// TIA Portal project "Encoder _3" (V16)

(* hardware
DEVICE "S7-1200 station_1"  S7-1200 Station
   slot 0: "Rack_0"  S7-1200 Rack  Rack  V1.0
   slot 1: "PLC_1"  CPU 1212C DC/DC/DC  6ES7 212-1AE40-0XB0  V4.1
*)

// ===== PLC "PLC_1"  CPU 1212C DC/DC/DC =====

VAR_GLOBAL   // PLC tag table "Default tag table"
   "System_Byte" AT %MD2 : DInt;
   "FirstScan" AT %M1.0 : Bool;
   "DiagStatusUpdate" AT %M1.1 : Bool;
   "AlwaysTRUE" AT %M1.2 : Bool;
   "AlwaysFALSE" AT %M1.3 : Bool;
   "Clock_Byte" AT %MB0 : Byte;
   "Clock_10Hz" AT %M0.0 : Bool;
   "Clock_5Hz" AT %M0.1 : Bool;
   "Clock_2.5Hz" AT %M0.2 : Bool;
   "Clock_2Hz" AT %M0.3 : Bool;
   "Clock_1.25Hz" AT %M0.4 : Bool;
   "Clock_1Hz" AT %M0.5 : Bool;
   "Clock_0.625Hz" AT %M0.6 : Bool;
   "Clock_0.5Hz" AT %M0.7 : Bool;
   "encoder" AT %ID1000 : DInt;
   "Tag_2" AT %Q0.0 : Bool;
   "al_limite_atg" AT %Q0.1 : Bool;
   "Tag_4" AT %Q0.3 : Bool;
   "Tag_5" AT %I0.0 : Bool;
   "Tag_6" AT %I0.1 : Bool;
   "Tag_7" AT %I0.2 : Bool;
   "clock" AT %M255.5 : Bool;
   "time_et" AT %MD256 : Time;
   "numero_rotacao" AT %MW300 : Word;
   "time_pt" AT %MD200 : Time;
   "Tag_1" AT %ID100 : DWord;
END_VAR

VAR_GLOBAL   // PLC tag table "Tag table_1"
   "SLI_DETACH_event" AT %I0.3 : Bool;
END_VAR

TYPE "User_data_type_1"
   STRUCT
      Element_1 : Bool;
   END_STRUCT;
END_TYPE

DATA_BLOCK "Data_block_1"   // DB1
{ S7_Optimized_Access := 'TRUE' }
VERSION : 0.1
   VAR RETAIN
      valor_contagem : DInt;
   END_VAR
   VAR
      valor_referencia : DInt := 400;
      novo_valor : DInt;
   END_VAR
BEGIN
END_DATA_BLOCK

ORGANIZATION_BLOCK "Main"   // OB1, LAD, ProgramCycle
TITLE = "Main Program Sweep (Cycle)"
{ S7_Optimized_Access := 'TRUE' }
VERSION : 0.1
   VAR_INPUT
      Initial_Call : Bool;   // Initial call of this OB
      Remanence : Bool;   // =True, if remanent data are available
   END_VAR
   VAR_TEMP
      Temp_1 : DInt;
   END_VAR
   VAR CONSTANT
      numero_rotacao : DInt;
   END_VAR
BEGIN

REGION Network 1
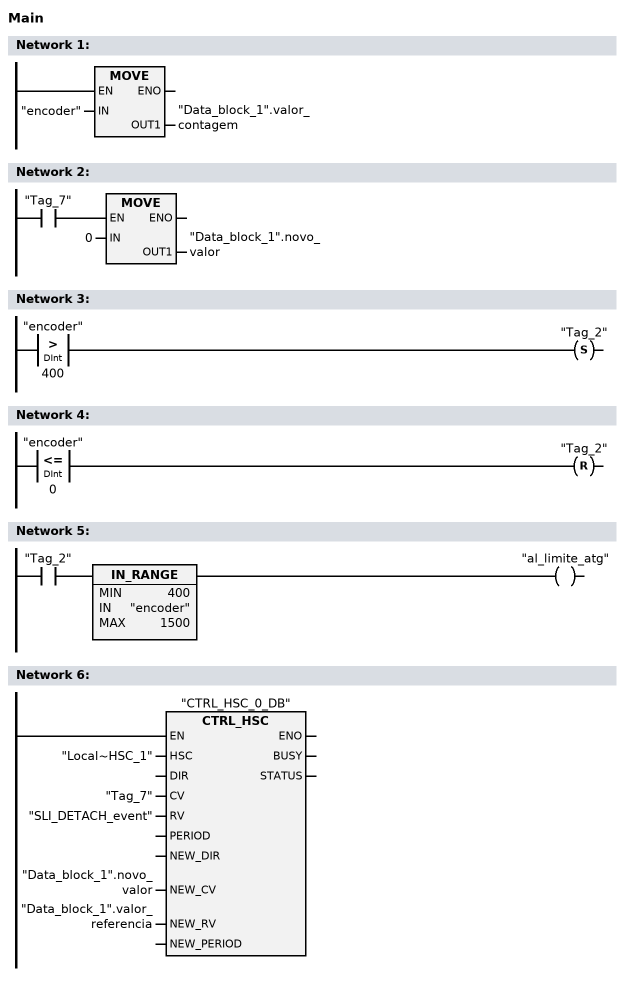
   RUNG wire#powerrail
      Move(in := "encoder", out1 => "Data_block_1".valor_contagem)
   END_RUNG
   // the same network as SCL:
   "Data_block_1".valor_contagem := "encoder";
END_REGION

REGION Network 2
   RUNG wire#powerrail
      Contact( "Tag_7" )
      Move(in := 0, out1 => "Data_block_1".novo_valor)
   END_RUNG
   // the same network as SCL:
   IF "Tag_7" THEN "Data_block_1".novo_valor := 0; END_IF;
END_REGION

REGION Network 3
   RUNG wire#powerrail
      { S7_Templates := "SrcType := DInt" } GT_Contact(in1 := "encoder", in2 := 400)
      S_Coil( "Tag_2" )
   END_RUNG
   // the same network as SCL:
   IF "encoder" > 400 THEN "Tag_2" := TRUE; END_IF;
END_REGION

REGION Network 4
   RUNG wire#powerrail
      { S7_Templates := "SrcType := DInt" } LE_Contact(in1 := "encoder", in2 := 0)
      R_Coil( "Tag_2" )
   END_RUNG
   // the same network as SCL:
   IF "encoder" <= 0 THEN "Tag_2" := FALSE; END_IF;
END_REGION

REGION Network 5
   RUNG wire#powerrail
      Contact( "Tag_2" )
      { S7_Templates := "SrcType := DInt" } InRange(min := 400, in := "encoder", max := 1500)
      Coil( "al_limite_atg" )
   END_RUNG
   // the same network as SCL:
   "al_limite_atg" := "Tag_2" AND (400 <= "encoder") AND ("encoder" <= 1500);
END_REGION

REGION Network 6
   "CTRL_HSC_0_DB"(HSC := "Local~HSC_1",   // CTRL_HSC
                   CV := "Tag_7",
                   RV := "SLI_DETACH_event",
                   NEW_CV := "Data_block_1".novo_valor,
                   NEW_RV := "Data_block_1".valor_referencia);
END_REGION
END_ORGANIZATION_BLOCK